# EPICS autosave request: xx_auto_icbAdc_settings.req
$(P)$(A)GAIN
$(P)$(A)OFFSET
$(P)$(A)AMOD
$(P)$(A)CMOD
$(P)$(A)LLD
$(P)$(A)ULD
$(P)$(A)ZERO
$(P)$(A)PMOD
$(P)$(A)GMOD
$(P)$(A)TMOD
